{attribute 'qualified_only'}
{attribute 'strict'}
TYPE E_HESULT_AdsErr :
(
	ERR_INTERNAL 				:= UDINT_TO_DINT((16#98110000 + 16#1)),		// Internal error.
	ERR_TARGETPORTNOTFOUND 		:= UDINT_TO_DINT((16#98110000 + 16#6)),		// Target port not found – ADS server is not started or is not reachable.
	ERR_TARGETMACHINENOTFOUND 	:= UDINT_TO_DINT((16#98110000 + 16#7)),		// Target computer not found – AMS route was not found. 
	ERR_PORTNOTCONNECTED		:= UDINT_TO_DINT((16#98110000 + 16#D)),		// Port not connected.
	ERR_INVALIDAMSLENGTH		:= UDINT_TO_DINT((16#98110000 + 16#E)),		// Invalid AMS length.
	ERR_INVALIDAMSNETID			:= UDINT_TO_DINT((16#98110000 + 16#F))		// Invalid AMS Net ID.
) DINT;
END_TYPE
//  ERR_INTERNAL = 'UDINT_TO_DINT((16#98110000 + 16#1))'
//  ERR_TARGETPORTNOTFOUND = 'UDINT_TO_DINT((16#98110000 + 16#6))'
//  ERR_TARGETMACHINENOTFOUND = 'UDINT_TO_DINT((16#98110000 + 16#7))'
//  ERR_PORTNOTCONNECTED = 'UDINT_TO_DINT((16#98110000 + 16#D))'
//  ERR_INVALIDAMSLENGTH = 'UDINT_TO_DINT((16#98110000 + 16#E))'
//  ERR_INVALIDAMSNETID = 'UDINT_TO_DINT((16#98110000 + 16#F))'

(* stored: Version 1.1.0.1, ProductVersion 3.1.4026.18
   EnumerationTextList E_HESULT_AdsErr: Id {b04bf851-5b9e-4948-a5dc-53f5178e2761} *)
